FUNCTION_BLOCK CLOCK_PLS
VAR_INPUT
	bCpStart			: BOOL;
	INT_TIME_ms 	: INT;

END_VAR
VAR_OUTPUT
	CLOCK_PLS_BOOL: BOOL;
END_VAR
VAR
	T0: TON;
	T1: TON;
	M0: BOOL;
	M1: BOOL;
	D0: TIME;
	D1: TIME;
END_VAR

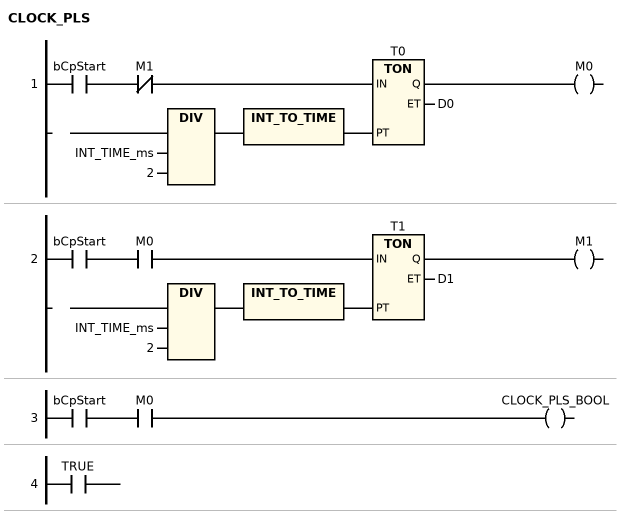
// NETWORK 1
T0(IN := bCpStart AND NOT M1, PT := INT_TO_TIME(INT_TIME_ms / 2), ET => D0); // TON
M0 := T0.Q;

// NETWORK 2
T1(IN := bCpStart AND M0, PT := INT_TO_TIME(INT_TIME_ms / 2), ET => D1); // TON
M1 := T1.Q;

// NETWORK 3
CLOCK_PLS_BOOL := bCpStart AND M0;

// NETWORK 4

END_FUNCTION_BLOCK

(* stored: Version 1.1.0.1, ProductVersion 3.1.4024.12
   POU CLOCK_PLS: Id {6b39117d-12de-4709-9d45-45e810bb21f1}, SpecialFunc None *)
